{attribute 'qualified_only'}
VAR_GLOBAL
	TxBuffer: ComBuffer;
	RxBuffer: ComBuffer;
END_VAR

(* stored: Version 1.1.0.1, ProductVersion 3.1.4024.11
   GVL GVL: Id {462252f0-b561-4319-8428-9d34ba2b3770} *)
